{attribute 'c++_compatible'}
FUNCTION_BLOCK TransportSystem EXTENDS TcBaseModuleRegistered IMPLEMENTS I_Transport
VAR_INPUT
END_VAR
VAR_OUTPUT
END_VAR
VAR		
	// ===== Motion Control =====
	fbMc_MoveVelocity: MC_MoveVelocity;	// continous motion
	fbMc_Stop: MC_Stop;					// stop
	fbMc_Power: MC_Power;				// power
	axisTransportA: AXIS_REF;			// Master axis
	
	// ==== States ====
	eZustand: E_STATES := E_STATES.Stopped;	// aktueller Zustand
	//bRunning: BOOL := FALSE;
	bReady: BOOL := FALSE;				// Achse bereit?
	rVelocity: LREAL;					// Velocity
	
	// ==== Outputs ====
	rActVelocity AT %Q*: LREAL;				// Actual Velocity output
END_VAR

// ==== Inputs ====
axisTransportA.ReadStatus();

// ==== Outputs ====
// aktuelle Geschwindigkeit
rActVelocity := axisTransportA.NcToPlc.ActVelo;

// ==== Statemachine ====
CASE eZustand OF
	E_STATES.Starting:
		THIS^.Starting();

	E_STATES.Started:
		// idle
	
	E_STATES.Stopping:
		THIS^.Stopping();
	
	E_STATES.Stopped:
		// idle
	
END_CASE

METHOD FB_reinit : BOOL
VAR_INPUT
END_VAR
SUPER^.FB_reinit();
END_METHOD

{attribute 'TcTypeSystem'}
{attribute 'no-analysis'}
{attribute 'c++_compatible'}
{attribute 'minimal_input_size' := '4'}
{attribute 'pack_mode' := '4'}
METHOD Start : HRESULT
VAR_INPUT
	rVelocity : LREAL;
END_VAR
THIS^.rVelocity := rVelocity;

eZustand := E_STATES.Starting;

bReady := FALSE;
END_METHOD

METHOD Starting : BOOL
VAR_INPUT
END_VAR
// Achse starten und wenn Sie bereit ist, auf gegebene Geschwindigkeit ziehen
// MC_POWER -> MC_MoveVelocity

// TODO jeden Baustein auf Fehler prüfen, evtl allgemeinen Zustand Error einführen

// Achse ist nicht bereit (nicht mit MC_Power freigegeben)
IF NOT bReady THEN
	fbMc_Power(
		Axis := axisTransportA,
		Enable := TRUE,
		Enable_Positive := TRUE,
		Status => bReady
	);
ELSE // Achse ist bereit und beschleunigt auf Zielgeschwindigkeit
	fbMc_MoveVelocity(
		Execute := TRUE,
		Axis := axisTransportA,
		Direction := MC_Direction.MC_Positive_Direction,
		Velocity := rVelocity
	);

	// Achse hat Zielgeschwindigkeit erreicht => Zustand: Started
	IF fbMc_MoveVelocity.InVelocity THEN
		THIS^.eZustand := E_STATES.Started;
	END_IF	
END_IF


// TODO IF fbMc_Power.Error THEN ... log Error Event + Zustand: Error
END_METHOD

{attribute 'TcTypeSystem'}
{attribute 'no-analysis'}
{attribute 'c++_compatible'}
{attribute 'minimal_input_size' := '4'}
{attribute 'pack_mode' := '4'}
METHOD Stop : HRESULT
eZustand := E_STATES.Stopping;
END_METHOD

METHOD PRIVATE Stopping : BOOL
VAR_INPUT
END_VAR
fbMc_MoveVelocity(
	Axis := axisTransportA,
	Execute := FALSE
);

fbMc_Stop(
	Axis := axisTransportA,
	Execute := TRUE
);

IF fbMc_Stop.Done THEN
	bReady := FALSE;
	// Nach Stop, Achse wieder durch Execute := FALSE entriegeln
	fbMc_Stop(
		Axis := axisTransportA,
		Execute := FALSE
	);
	eZustand := E_STATES.Stopped;
END_IF
END_METHOD

{attribute 'TcTypeSystem'}
{attribute 'no-analysis'}
{attribute 'c++_compatible'}
{attribute 'minimal_input_size' := '4'}
{attribute 'pack_mode' := '4'}
METHOD TcQueryInterface : HRESULT
VAR_INPUT
	iid	: REFERENCE TO IID;
	pipItf	: POINTER TO PVOID;
END_VAR
VAR
	ipTPS: I_Transport;
END_VAR
IF GuidsEqual(ADR(iid), ADR(TC_GLOBAL_IID_LIST.IID_I_Transport)) THEN
	ipTPS := THIS^;
	pipItf^ := ITCUNKNOWN_TO_PVOID(ipTPS);
	TcAddRef();
	TcQueryInterface := S_OK;
ELSE
	TcQueryInterface := SUPER^.TcQueryInterface(iid, pipItf);
END_IF
END_METHOD

END_FUNCTION_BLOCK

(* stored: Version 1.1.0.1, ProductVersion 3.1.4024.3
   POU TransportSystem: Id {c996a55c-9379-43f7-b519-663e18e9a46c}, SpecialFunc None
   Method FB_reinit: Id {d6424f74-746a-4e64-95f1-809deeaadf5b}
   Method Start: Id {81a3c96c-a6ad-4da3-a672-eeb93b9b90af}
   Method Starting: Id {93cbcf18-b403-4866-a1fc-9eb7c910d004}
   Method Stop: Id {da4e9d46-829c-4842-a396-f09d476ba41f}
   Method Stopping: Id {8d6ba368-5131-4c7f-91ad-3948674802b2}
   Method TcQueryInterface: Id {ef707d13-eddd-40e5-8339-1abf15b0f049} *)
